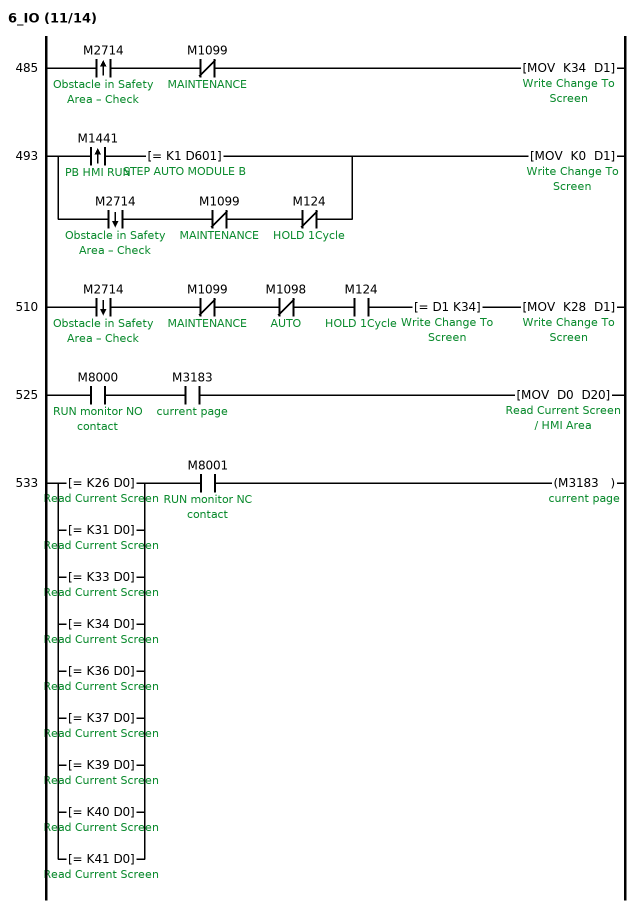
[picture p72: ladder of 6_IO, rungs at steps 485 to 533]
485   LDP     M2714  ; Obstacle in Safety Area – Check
      ANI     M1099  ; MAINTENANCE
      MOV     K34 D1  ; Write Change To Screen
493   LDP     M1441  ; PB HMI RUN
      AND=    K1 D601  ; STEP AUTO MODULE B
      LDF     M2714  ; Obstacle in Safety Area – Check
      ANI     M1099  ; MAINTENANCE
      ANI     M124  ; HOLD 1Cycle
      ORB
      MOV     K0 D1
510   LDF     M2714  ; Obstacle in Safety Area – Check
      ANI     M1099  ; MAINTENANCE
      ANI     M1098  ; AUTO
      AND     M124  ; HOLD 1Cycle
      AND=    D1 K34  ; Write Change To Screen
      MOV     K28 D1
525   LD      M8000  ; RUN monitor NO contact
      AND     M3183  ; current page
      MOV     D0 D20  ; Read Current Screen / HMI Area
533   LD=     K26 D0  ; Read Current Screen
      OR=     K31 D0  ; Read Current Screen
      OR=     K33 D0  ; Read Current Screen
      OR=     K34 D0  ; Read Current Screen
      OR=     K36 D0  ; Read Current Screen
      OR=     K37 D0  ; Read Current Screen
      OR=     K39 D0  ; Read Current Screen
      OR=     K40 D0  ; Read Current Screen
      OR=     K41 D0  ; Read Current Screen
      AND     M8001  ; RUN monitor NC contact
      OUT     M3183  ; current page
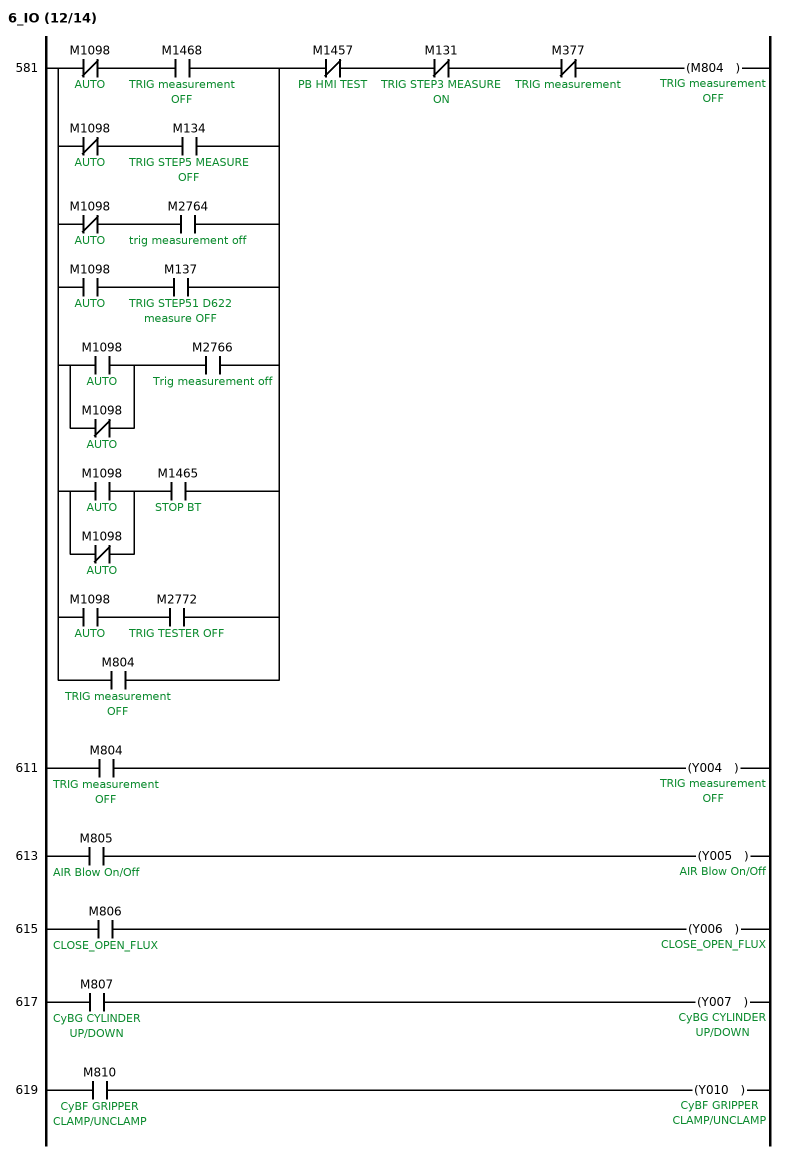
581   LDI     M1098  ; AUTO
      AND     M1468  ; TRIG measurement OFF
      LDI     M1098  ; AUTO
      AND     M134  ; TRIG STEP5 MEASURE OFF
      ORB
      LDI     M1098  ; AUTO
      AND     M2764  ; trig measurement off
      ORB
      LD      M1098  ; AUTO
      AND     M137  ; TRIG STEP51 D622 measure OFF
      ORB
      LD      M1098  ; AUTO
      ORI     M1098  ; AUTO
      AND     M2766  ; Trig measurement off
      ORB
      LD      M1098  ; AUTO
      ORI     M1098  ; AUTO
      AND     M1465  ; STOP BT
      ORB
      LD      M1098  ; AUTO
      AND     M2772  ; TRIG TESTER OFF
      ORB
      OR      M804  ; TRIG measurement OFF
      ANI     M1457  ; PB HMI TEST
      ANI     M131  ; TRIG STEP3 MEASURE ON
      ANI     M377  ; TRIG measurement
      OUT     M804  ; TRIG measurement OFF
611   LD      M804  ; TRIG measurement OFF
      OUT     Y004  ; TRIG measurement OFF
613   LD      M805  ; AIR Blow On/Off
      OUT     Y005  ; AIR Blow On/Off
615   LD      M806  ; CLOSE_OPEN_FLUX
      OUT     Y006  ; CLOSE_OPEN_FLUX
617   LD      M807  ; CyBG CYLINDER UP/DOWN
      OUT     Y007  ; CyBG CYLINDER UP/DOWN
619   LD      M810  ; CyBF GRIPPER CLAMP/UNCLAMP
      OUT     Y010  ; CyBF GRIPPER CLAMP/UNCLAMP
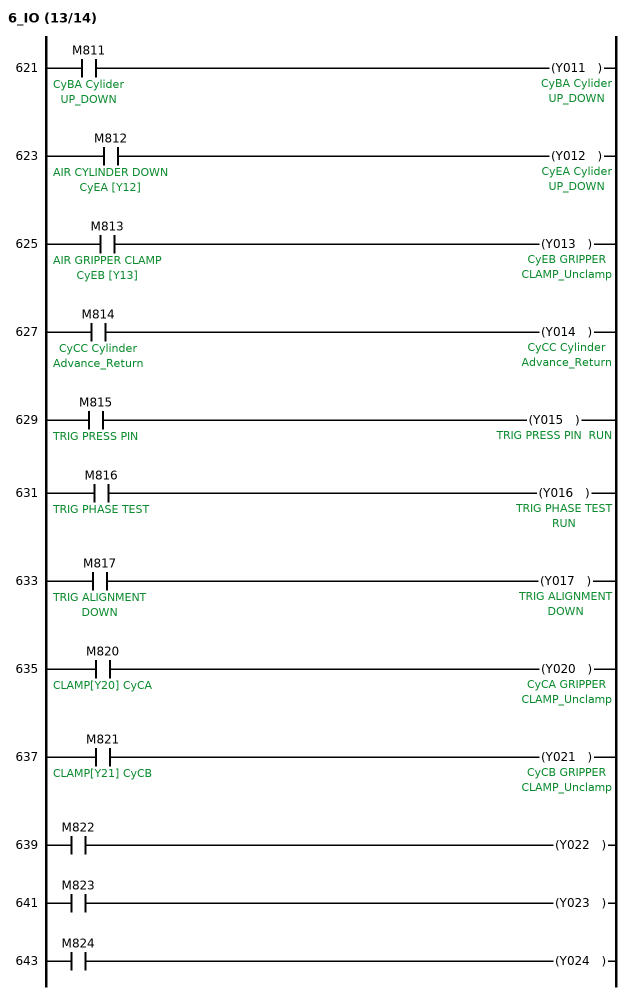
621   LD      M811  ; CyBA Cylider UP_DOWN
      OUT     Y011  ; CyBA Cylider UP_DOWN
623   LD      M812  ; AIR CYLINDER DOWN CyEA [Y12]
      OUT     Y012  ; CyEA Cylider UP_DOWN
625   LD      M813  ; AIR GRIPPER CLAMP CyEB [Y13]
      OUT     Y013  ; CyEB GRIPPER CLAMP_Unclamp
627   LD      M814  ; CyCC Cylinder Advance_Return
      OUT     Y014  ; CyCC Cylinder Advance_Return
629   LD      M815  ; TRIG PRESS PIN
      OUT     Y015  ; TRIG PRESS PIN  RUN
631   LD      M816  ; TRIG PHASE TEST
      OUT     Y016  ; TRIG PHASE TEST  RUN
633   LD      M817  ; TRIG ALIGNMENT  DOWN
      OUT     Y017  ; TRIG ALIGNMENT  DOWN
635   LD      M820  ; CLAMP[Y20] CyCA
      OUT     Y020  ; CyCA GRIPPER CLAMP_Unclamp
637   LD      M821  ; CLAMP[Y21] CyCB
      OUT     Y021  ; CyCB GRIPPER CLAMP_Unclamp
639   LD      M822
      OUT     Y022
641   LD      M823
      OUT     Y023
643   LD      M824
      OUT     Y024
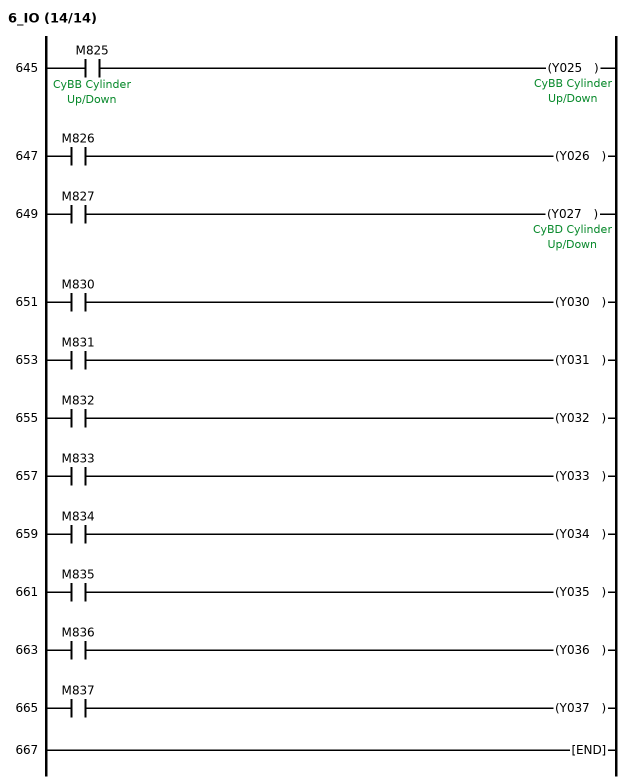
645   LD      M825  ; CyBB Cylinder Up/Down
      OUT     Y025  ; CyBB Cylinder Up/Down
647   LD      M826
      OUT     Y026
649   LD      M827
      OUT     Y027  ; CyBD Cylinder Up/Down
651   LD      M830
      OUT     Y030
653   LD      M831
      OUT     Y031
655   LD      M832
      OUT     Y032
657   LD      M833
      OUT     Y033
659   LD      M834
      OUT     Y034
661   LD      M835
      OUT     Y035
663   LD      M836
      OUT     Y036
665   LD      M837
      OUT     Y037
667   END
END_PROGRAM

PROGRAM 7_ALARM
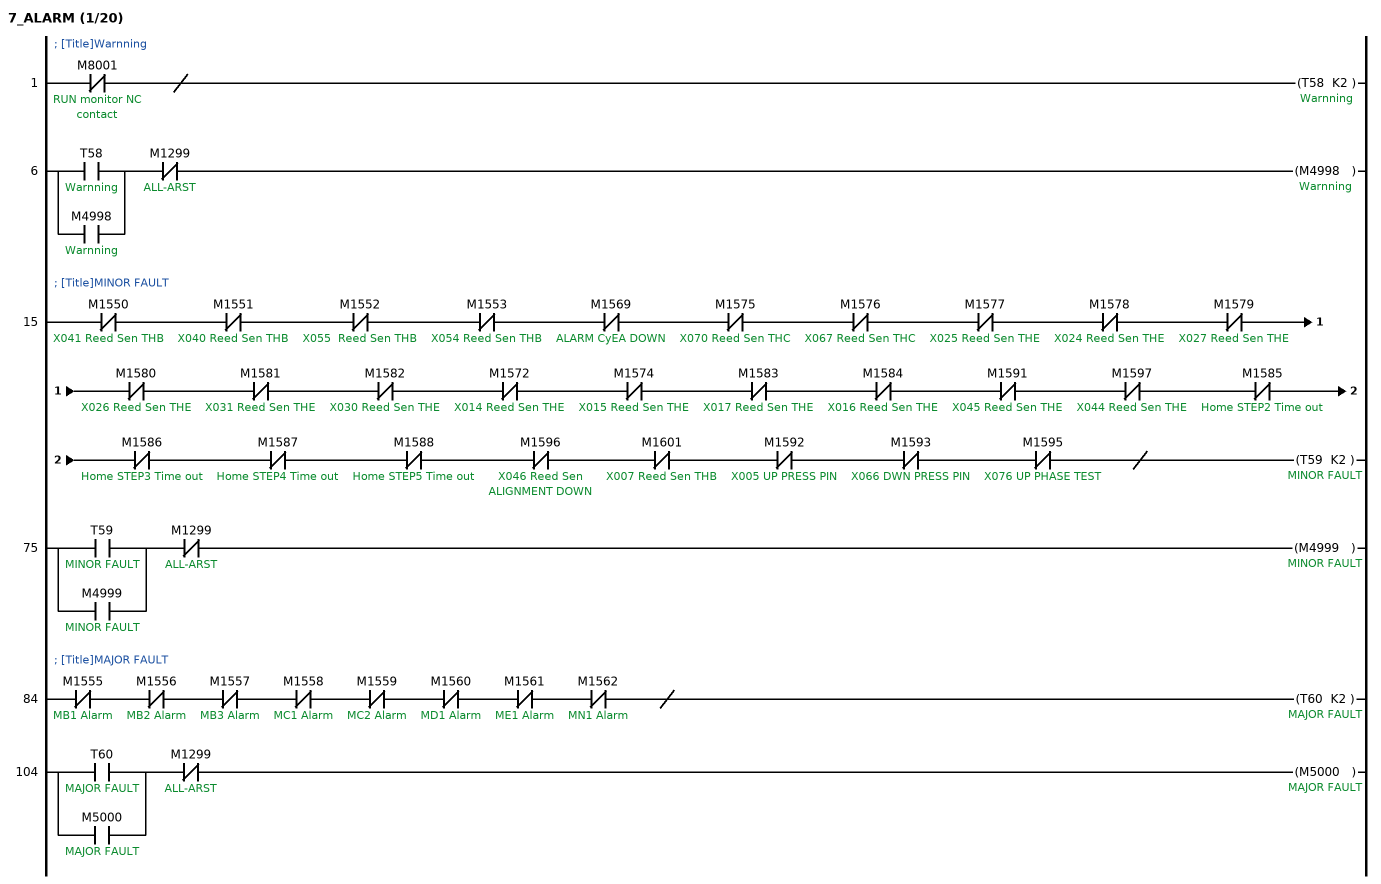
; [Title]Warnning
1     LDI     M8001  ; RUN monitor NC contact
      INV
      OUT     T58 K2  ; Warnning
6     LD      T58  ; Warnning
      OR      M4998  ; Warnning
      ANI     M1299  ; ALL-ARST
      OUT     M4998  ; Warnning
; [Title]MINOR FAULT
15    LDI     M1550  ; X041 Reed Sen THB
      ANI     M1551  ; X040 Reed Sen THB
      ANI     M1552  ; X055  Reed Sen THB
      ANI     M1553  ; X054 Reed Sen THB
      ANI     M1569  ; ALARM CyEA DOWN
      ANI     M1575  ; X070 Reed Sen THC
      ANI     M1576  ; X067 Reed Sen THC
      ANI     M1577  ; X025 Reed Sen THE
      ANI     M1578  ; X024 Reed Sen THE
      ANI     M1579  ; X027 Reed Sen THE
      ANI     M1580  ; X026 Reed Sen THE
      ANI     M1581  ; X031 Reed Sen THE
      ANI     M1582  ; X030 Reed Sen THE
      ANI     M1572  ; X014 Reed Sen THE
      ANI     M1574  ; X015 Reed Sen THE
      ANI     M1583  ; X017 Reed Sen THE
      ANI     M1584  ; X016 Reed Sen THE
      ANI     M1591  ; X045 Reed Sen THE
      ANI     M1597  ; X044 Reed Sen THE
      ANI     M1585  ; Home STEP2 Time out
      ANI     M1586  ; Home STEP3 Time out
      ANI     M1587  ; Home STEP4 Time out
      ANI     M1588  ; Home STEP5 Time out
      ANI     M1596  ; X046 Reed Sen ALIGNMENT DOWN
      ANI     M1601  ; X007 Reed Sen THB
      ANI     M1592  ; X005 UP PRESS PIN
      ANI     M1593  ; X066 DWN PRESS PIN
      ANI     M1595  ; X076 UP PHASE TEST
      INV
      OUT     T59 K2  ; MINOR FAULT
75    LD      T59  ; MINOR FAULT
      OR      M4999  ; MINOR FAULT
      ANI     M1299  ; ALL-ARST
      OUT     M4999  ; MINOR FAULT
; [Title]MAJOR FAULT
84    LDI     M1555  ; MB1 Alarm
      ANI     M1556  ; MB2 Alarm
      ANI     M1557  ; MB3 Alarm
      ANI     M1558  ; MC1 Alarm
      ANI     M1559  ; MC2 Alarm
      ANI     M1560  ; MD1 Alarm
      ANI     M1561  ; ME1 Alarm
      ANI     M1562  ; MN1 Alarm
      INV
      OUT     T60 K2  ; MAJOR FAULT
104   LD      T60  ; MAJOR FAULT
      OR      M5000  ; MAJOR FAULT
      ANI     M1299  ; ALL-ARST
      OUT     M5000  ; MAJOR FAULT
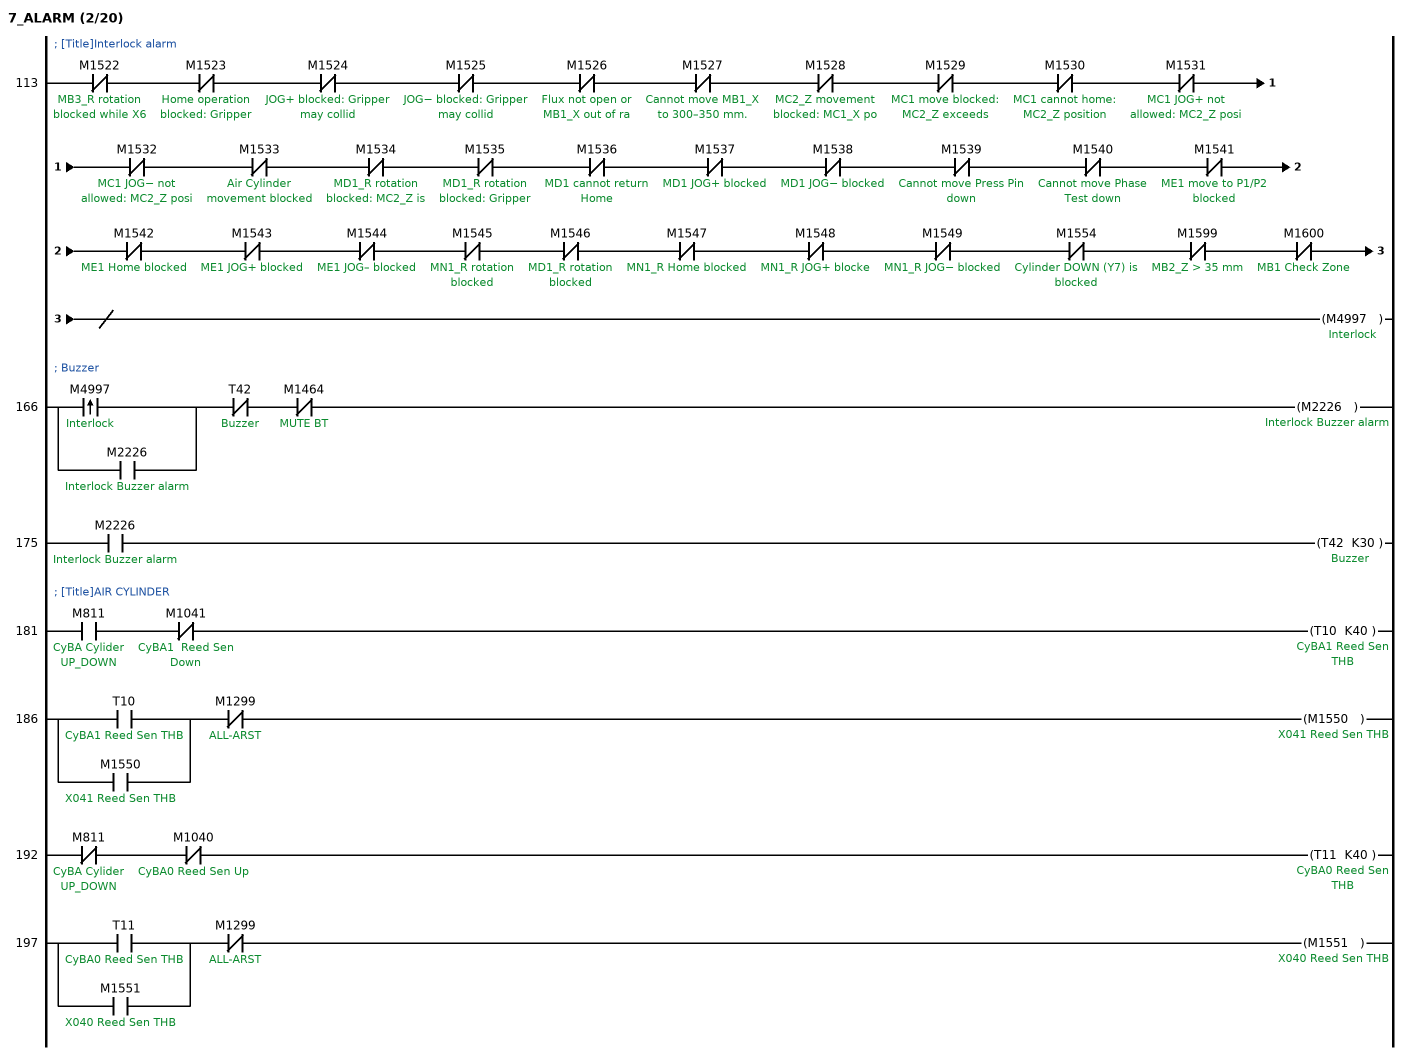
; [Title]Interlock alarm
113   LDI     M1522  ; MB3_R rotation blocked while X6
      ANI     M1523  ; Home operation blocked: Gripper
      ANI     M1524  ; JOG+ blocked: Gripper may collid
      ANI     M1525  ; JOG− blocked: Gripper may collid
      ANI     M1526  ; Flux not open or MB1_X out of ra
      ANI     M1527  ; Cannot move MB1_X to 300–350 mm.
      ANI     M1528  ; MC2_Z movement blocked: MC1_X po
      ANI     M1529  ; MC1 move blocked: MC2_Z exceeds
      ANI     M1530  ; MC1 cannot home: MC2_Z position
      ANI     M1531  ; MC1 JOG+ not allowed: MC2_Z posi
      ANI     M1532  ; MC1 JOG− not allowed: MC2_Z posi
      ANI     M1533  ; Air Cylinder movement blocked
      ANI     M1534  ; MD1_R rotation blocked: MC2_Z is
      ANI     M1535  ; MD1_R rotation blocked: Gripper
      ANI     M1536  ; MD1 cannot return Home
      ANI     M1537  ; MD1 JOG+ blocked
      ANI     M1538  ; MD1 JOG− blocked
      ANI     M1539  ; Cannot move Press Pin down
      ANI     M1540  ; Cannot move Phase Test down
      ANI     M1541  ; ME1 move to P1/P2 blocked
      ANI     M1542  ; ME1 Home blocked
      ANI     M1543  ; ME1 JOG+ blocked
      ANI     M1544  ; ME1 JOG– blocked
      ANI     M1545  ; MN1_R rotation blocked
      ANI     M1546  ; MD1_R rotation blocked
      ANI     M1547  ; MN1_R Home blocked
      ANI     M1548  ; MN1_R JOG+ blocke
      ANI     M1549  ; MN1_R JOG− blocked
      ANI     M1554  ; Cylinder DOWN (Y7) is blocked
      ANI     M1599  ; MB2_Z > 35 mm
      ANI     M1600  ; MB1 Check Zone
      INV
      OUT     M4997  ; Interlock
; Buzzer
166   LDP     M4997  ; Interlock
      OR      M2226  ; Interlock Buzzer alarm
      ANI     T42  ; Buzzer
      ANI     M1464  ; MUTE BT
      OUT     M2226  ; Interlock Buzzer alarm
175   LD      M2226  ; Interlock Buzzer alarm
      OUT     T42 K30  ; Buzzer
; [Title]AIR CYLINDER
181   LD      M811  ; CyBA Cylider UP_DOWN
      ANI     M1041  ; CyBA1  Reed Sen Down
      OUT     T10 K40  ; CyBA1 Reed Sen THB
186   LD      T10  ; CyBA1 Reed Sen THB
      OR      M1550  ; X041 Reed Sen THB
      ANI     M1299  ; ALL-ARST
      OUT     M1550  ; X041 Reed Sen THB
192   LDI     M811  ; CyBA Cylider UP_DOWN
      ANI     M1040  ; CyBA0 Reed Sen Up
      OUT     T11 K40  ; CyBA0 Reed Sen THB
197   LD      T11  ; CyBA0 Reed Sen THB
      OR      M1551  ; X040 Reed Sen THB
      ANI     M1299  ; ALL-ARST
      OUT     M1551  ; X040 Reed Sen THB
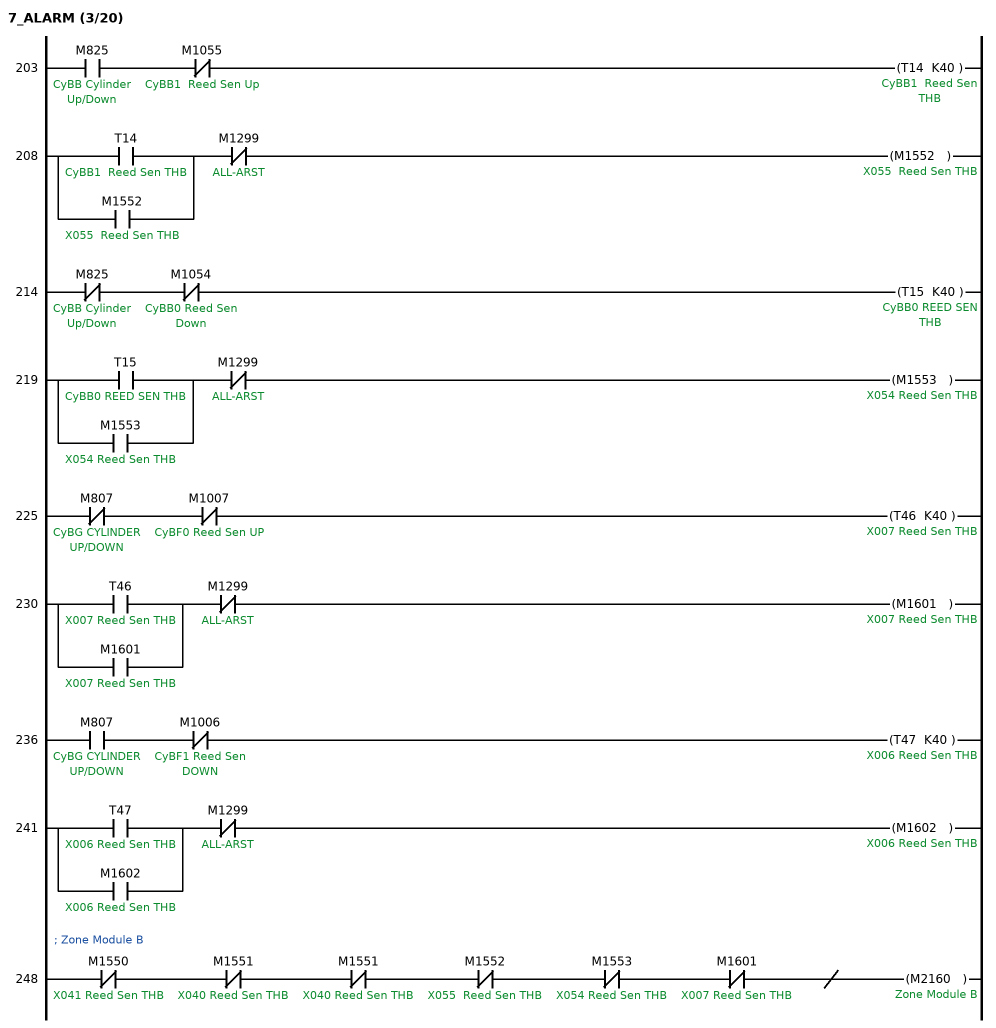
203   LD      M825  ; CyBB Cylinder Up/Down
      ANI     M1055  ; CyBB1  Reed Sen Up
      OUT     T14 K40  ; CyBB1  Reed Sen THB
208   LD      T14  ; CyBB1  Reed Sen THB
      OR      M1552  ; X055  Reed Sen THB
      ANI     M1299  ; ALL-ARST
      OUT     M1552  ; X055  Reed Sen THB
214   LDI     M825  ; CyBB Cylinder Up/Down
      ANI     M1054  ; CyBB0 Reed Sen Down
      OUT     T15 K40  ; CyBB0 REED SEN THB
219   LD      T15  ; CyBB0 REED SEN THB
      OR      M1553  ; X054 Reed Sen THB
      ANI     M1299  ; ALL-ARST
      OUT     M1553  ; X054 Reed Sen THB
225   LDI     M807  ; CyBG CYLINDER UP/DOWN
      ANI     M1007  ; CyBF0 Reed Sen UP
      OUT     T46 K40  ; X007 Reed Sen THB
230   LD      T46  ; X007 Reed Sen THB
      OR      M1601  ; X007 Reed Sen THB
      ANI     M1299  ; ALL-ARST
      OUT     M1601  ; X007 Reed Sen THB
236   LD      M807  ; CyBG CYLINDER UP/DOWN
      ANI     M1006  ; CyBF1 Reed Sen DOWN
      OUT     T47 K40  ; X006 Reed Sen THB
241   LD      T47  ; X006 Reed Sen THB
      OR      M1602  ; X006 Reed Sen THB
      ANI     M1299  ; ALL-ARST
      OUT     M1602  ; X006 Reed Sen THB
; Zone Module B
248   LDI     M1550  ; X041 Reed Sen THB
      ANI     M1551  ; X040 Reed Sen THB
      ANI     M1551  ; X040 Reed Sen THB
      ANI     M1552  ; X055  Reed Sen THB
      ANI     M1553  ; X054 Reed Sen THB
      ANI     M1601  ; X007 Reed Sen THB
      INV
      OUT     M2160  ; Zone Module B
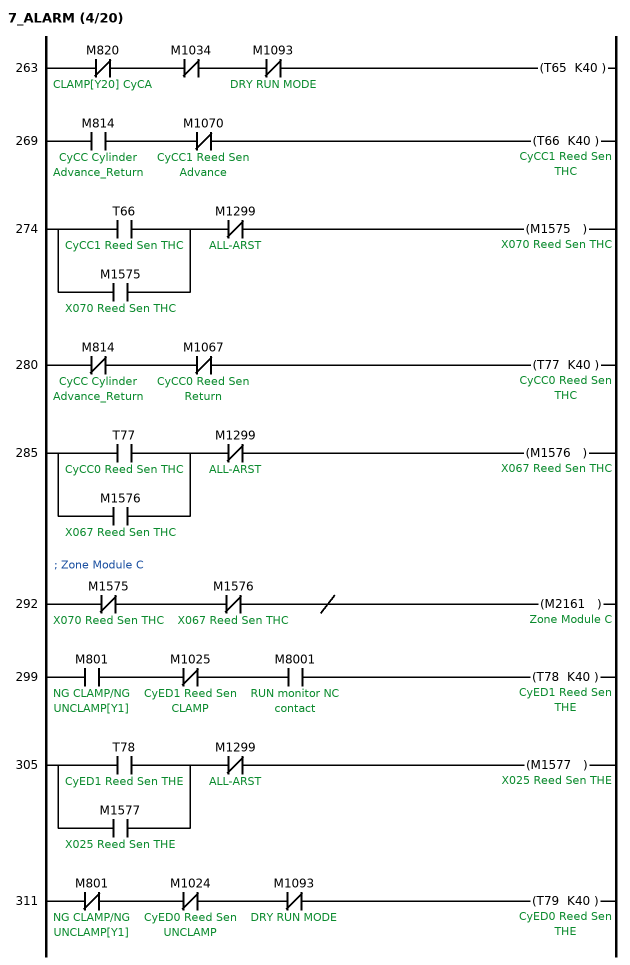
263   LDI     M820  ; CLAMP[Y20] CyCA
      ANI     M1034
      ANI     M1093  ; DRY RUN MODE
      OUT     T65 K40
269   LD      M814  ; CyCC Cylinder Advance_Return
      ANI     M1070  ; CyCC1 Reed Sen  Advance
      OUT     T66 K40  ; CyCC1 Reed Sen THC
274   LD      T66  ; CyCC1 Reed Sen THC
      OR      M1575  ; X070 Reed Sen THC
      ANI     M1299  ; ALL-ARST
      OUT     M1575  ; X070 Reed Sen THC
280   LDI     M814  ; CyCC Cylinder Advance_Return
      ANI     M1067  ; CyCC0 Reed Sen Return
      OUT     T77 K40  ; CyCC0 Reed Sen THC
285   LD      T77  ; CyCC0 Reed Sen THC
      OR      M1576  ; X067 Reed Sen THC
      ANI     M1299  ; ALL-ARST
      OUT     M1576  ; X067 Reed Sen THC
; Zone Module C
292   LDI     M1575  ; X070 Reed Sen THC
      ANI     M1576  ; X067 Reed Sen THC
      INV
      OUT     M2161  ; Zone Module C
299   LD      M801  ; NG CLAMP/NG UNCLAMP[Y1]
      ANI     M1025  ; CyED1 Reed Sen CLAMP
      AND     M8001  ; RUN monitor NC contact
      OUT     T78 K40  ; CyED1 Reed Sen THE
305   LD      T78  ; CyED1 Reed Sen THE
      OR      M1577  ; X025 Reed Sen THE
      ANI     M1299  ; ALL-ARST
      OUT     M1577  ; X025 Reed Sen THE
311   LDI     M801  ; NG CLAMP/NG UNCLAMP[Y1]
      ANI     M1024  ; CyED0 Reed Sen UNCLAMP
      ANI     M1093  ; DRY RUN MODE
      OUT     T79 K40  ; CyED0 Reed Sen THE
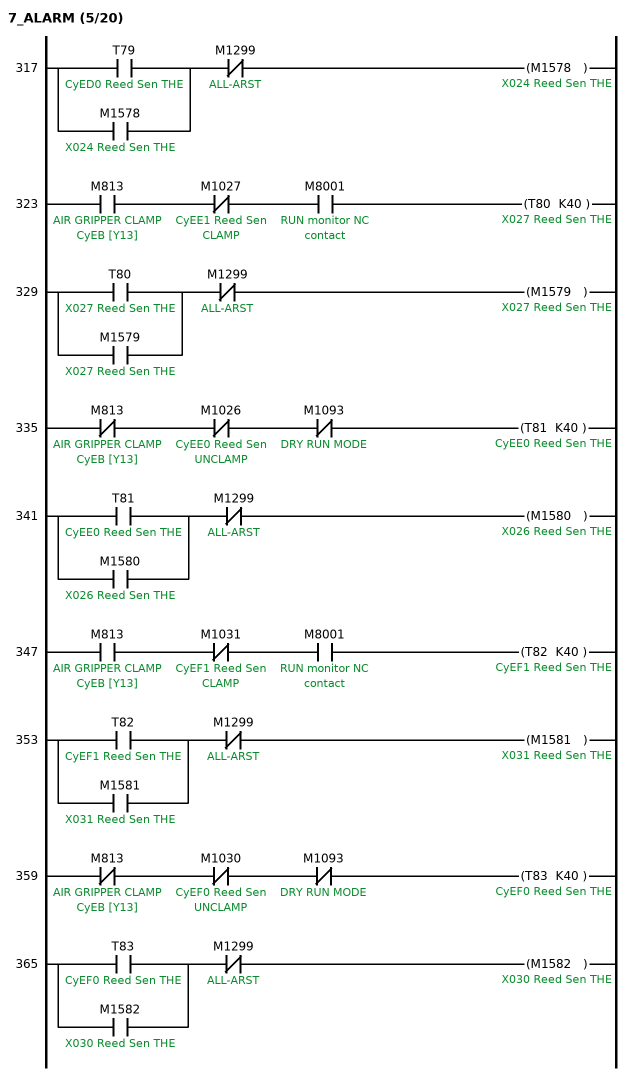
317   LD      T79  ; CyED0 Reed Sen THE
      OR      M1578  ; X024 Reed Sen THE
      ANI     M1299  ; ALL-ARST
      OUT     M1578  ; X024 Reed Sen THE
323   LD      M813  ; AIR GRIPPER CLAMP CyEB [Y13]
      ANI     M1027  ; CyEE1 Reed Sen CLAMP
      AND     M8001  ; RUN monitor NC contact
      OUT     T80 K40  ; X027 Reed Sen THE
329   LD      T80  ; X027 Reed Sen THE
      OR      M1579  ; X027 Reed Sen THE
      ANI     M1299  ; ALL-ARST
      OUT     M1579  ; X027 Reed Sen THE
335   LDI     M813  ; AIR GRIPPER CLAMP CyEB [Y13]
      ANI     M1026  ; CyEE0 Reed Sen UNCLAMP
      ANI     M1093  ; DRY RUN MODE
      OUT     T81 K40  ; CyEE0 Reed Sen THE
341   LD      T81  ; CyEE0 Reed Sen THE
      OR      M1580  ; X026 Reed Sen THE
      ANI     M1299  ; ALL-ARST
      OUT     M1580  ; X026 Reed Sen THE
347   LD      M813  ; AIR GRIPPER CLAMP CyEB [Y13]
      ANI     M1031  ; CyEF1 Reed Sen CLAMP
      AND     M8001  ; RUN monitor NC contact
      OUT     T82 K40  ; CyEF1 Reed Sen THE
353   LD      T82  ; CyEF1 Reed Sen THE
      OR      M1581  ; X031 Reed Sen THE
      ANI     M1299  ; ALL-ARST
      OUT     M1581  ; X031 Reed Sen THE
359   LDI     M813  ; AIR GRIPPER CLAMP CyEB [Y13]
      ANI     M1030  ; CyEF0 Reed Sen UNCLAMP
      ANI     M1093  ; DRY RUN MODE
      OUT     T83 K40  ; CyEF0 Reed Sen THE
365   LD      T83  ; CyEF0 Reed Sen THE
      OR      M1582  ; X030 Reed Sen THE
      ANI     M1299  ; ALL-ARST
      OUT     M1582  ; X030 Reed Sen THE
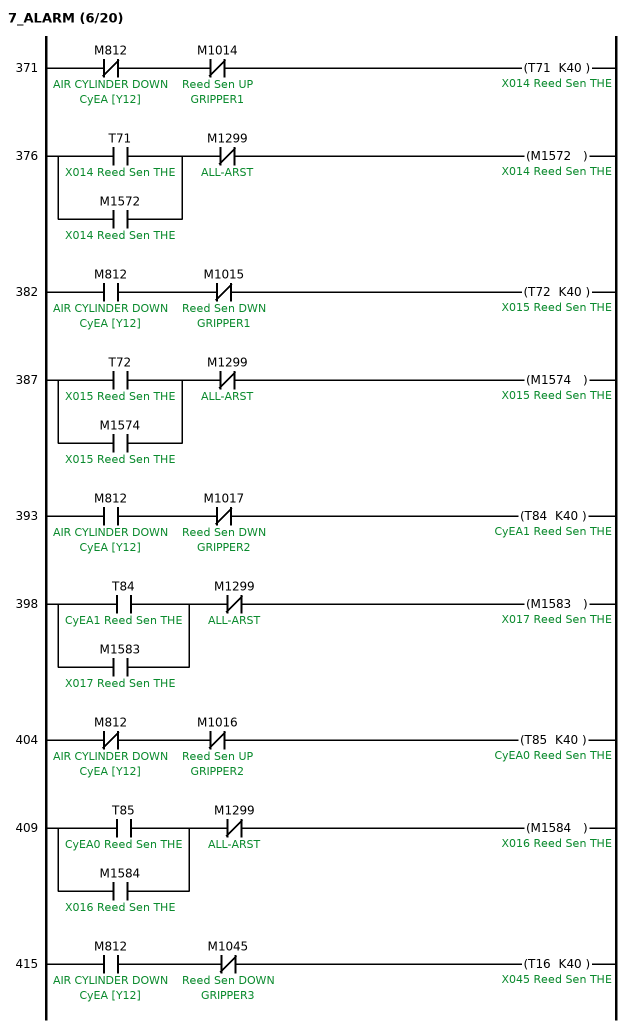
371   LDI     M812  ; AIR CYLINDER DOWN CyEA [Y12]
      ANI     M1014  ; Reed Sen UP GRIPPER1
      OUT     T71 K40  ; X014 Reed Sen THE
376   LD      T71  ; X014 Reed Sen THE
      OR      M1572  ; X014 Reed Sen THE
      ANI     M1299  ; ALL-ARST
      OUT     M1572  ; X014 Reed Sen THE
382   LD      M812  ; AIR CYLINDER DOWN CyEA [Y12]
      ANI     M1015  ; Reed Sen DWN GRIPPER1
      OUT     T72 K40  ; X015 Reed Sen THE
387   LD      T72  ; X015 Reed Sen THE
      OR      M1574  ; X015 Reed Sen THE
      ANI     M1299  ; ALL-ARST
      OUT     M1574  ; X015 Reed Sen THE
393   LD      M812  ; AIR CYLINDER DOWN CyEA [Y12]
      ANI     M1017  ; Reed Sen DWN GRIPPER2
      OUT     T84 K40  ; CyEA1 Reed Sen THE
398   LD      T84  ; CyEA1 Reed Sen THE
      OR      M1583  ; X017 Reed Sen THE
      ANI     M1299  ; ALL-ARST
      OUT     M1583  ; X017 Reed Sen THE
404   LDI     M812  ; AIR CYLINDER DOWN CyEA [Y12]
      ANI     M1016  ; Reed Sen UP GRIPPER2
      OUT     T85 K40  ; CyEA0 Reed Sen THE
409   LD      T85  ; CyEA0 Reed Sen THE
      OR      M1584  ; X016 Reed Sen THE
      ANI     M1299  ; ALL-ARST
      OUT     M1584  ; X016 Reed Sen THE
415   LD      M812  ; AIR CYLINDER DOWN CyEA [Y12]
      ANI     M1045  ; Reed Sen DOWN GRIPPER3
      OUT     T16 K40  ; X045 Reed Sen THE
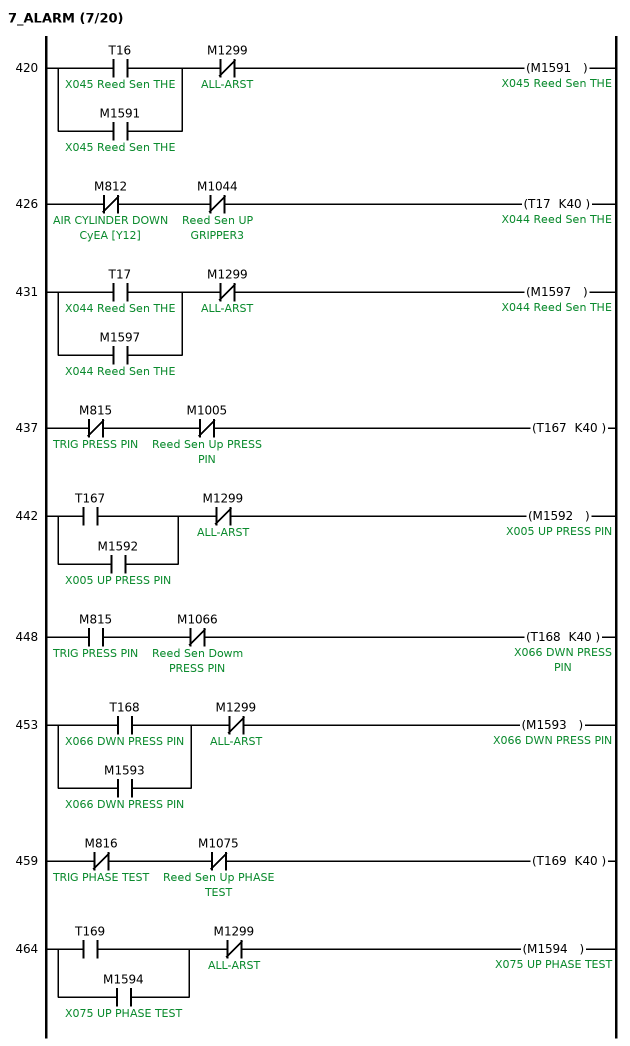
420   LD      T16  ; X045 Reed Sen THE
      OR      M1591  ; X045 Reed Sen THE
      ANI     M1299  ; ALL-ARST
      OUT     M1591  ; X045 Reed Sen THE
426   LDI     M812  ; AIR CYLINDER DOWN CyEA [Y12]
      ANI     M1044  ; Reed Sen UP GRIPPER3
      OUT     T17 K40  ; X044 Reed Sen THE
431   LD      T17  ; X044 Reed Sen THE
      OR      M1597  ; X044 Reed Sen THE
      ANI     M1299  ; ALL-ARST
      OUT     M1597  ; X044 Reed Sen THE
437   LDI     M815  ; TRIG PRESS PIN
      ANI     M1005  ; Reed Sen Up PRESS PIN
      OUT     T167 K40
442   LD      T167
      OR      M1592  ; X005 UP PRESS PIN
      ANI     M1299  ; ALL-ARST
      OUT     M1592  ; X005 UP PRESS PIN
448   LD      M815  ; TRIG PRESS PIN
      ANI     M1066  ; Reed Sen Dowm PRESS PIN
      OUT     T168 K40  ; X066 DWN PRESS PIN
453   LD      T168  ; X066 DWN PRESS PIN
      OR      M1593  ; X066 DWN PRESS PIN
      ANI     M1299  ; ALL-ARST
      OUT     M1593  ; X066 DWN PRESS PIN
459   LDI     M816  ; TRIG PHASE TEST
      ANI     M1075  ; Reed Sen Up PHASE TEST
      OUT     T169 K40
464   LD      T169
      OR      M1594  ; X075 UP PHASE TEST
      ANI     M1299  ; ALL-ARST
      OUT     M1594  ; X075 UP PHASE TEST
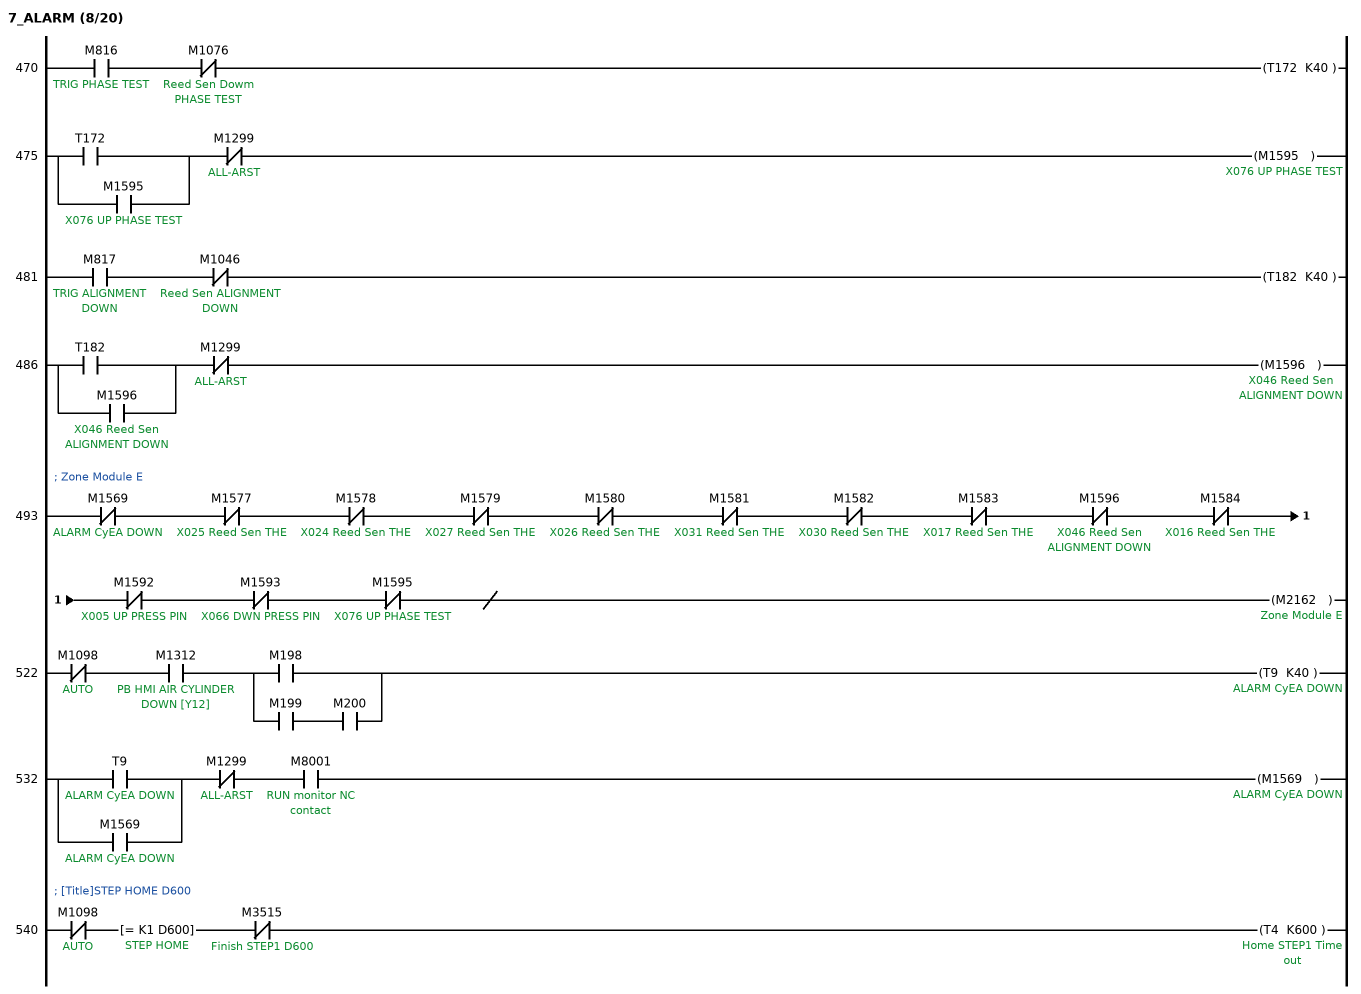
470   LD      M816  ; TRIG PHASE TEST
      ANI     M1076  ; Reed Sen Dowm PHASE TEST
      OUT     T172 K40
475   LD      T172
      OR      M1595  ; X076 UP PHASE TEST
      ANI     M1299  ; ALL-ARST
      OUT     M1595  ; X076 UP PHASE TEST
481   LD      M817  ; TRIG ALIGNMENT  DOWN
      ANI     M1046  ; Reed Sen ALIGNMENT DOWN
      OUT     T182 K40
486   LD      T182
      OR      M1596  ; X046 Reed Sen ALIGNMENT DOWN
      ANI     M1299  ; ALL-ARST
      OUT     M1596  ; X046 Reed Sen ALIGNMENT DOWN
; Zone Module E
493   LDI     M1569  ; ALARM CyEA DOWN
      ANI     M1577  ; X025 Reed Sen THE
      ANI     M1578  ; X024 Reed Sen THE
      ANI     M1579  ; X027 Reed Sen THE
      ANI     M1580  ; X026 Reed Sen THE
      ANI     M1581  ; X031 Reed Sen THE
      ANI     M1582  ; X030 Reed Sen THE
      ANI     M1583  ; X017 Reed Sen THE
      ANI     M1596  ; X046 Reed Sen ALIGNMENT DOWN
      ANI     M1584  ; X016 Reed Sen THE
      ANI     M1592  ; X005 UP PRESS PIN
      ANI     M1593  ; X066 DWN PRESS PIN
      ANI     M1595  ; X076 UP PHASE TEST
      INV
      OUT     M2162  ; Zone Module E
522   LDI     M1098  ; AUTO
      AND     M1312  ; PB HMI AIR CYLINDER DOWN [Y12]
      LD      M198
      LD      M199
      AND     M200
      ORB
      ANB
      OUT     T9 K40  ; ALARM CyEA DOWN
532   LD      T9  ; ALARM CyEA DOWN
      OR      M1569  ; ALARM CyEA DOWN
      ANI     M1299  ; ALL-ARST
      AND     M8001  ; RUN monitor NC contact
      OUT     M1569  ; ALARM CyEA DOWN
; [Title]STEP HOME D600
540   LDI     M1098  ; AUTO
      AND=    K1 D600  ; STEP HOME
      ANI     M3515  ; Finish STEP1 D600
      OUT     T4 K600  ; Home STEP1 Time out
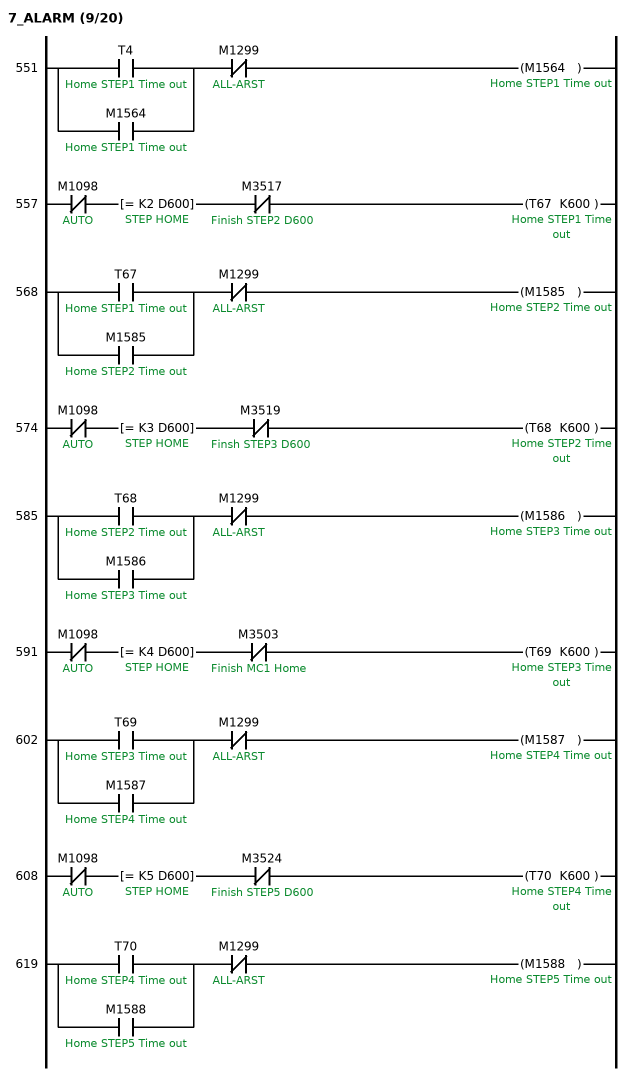
551   LD      T4  ; Home STEP1 Time out
      OR      M1564  ; Home STEP1 Time out
      ANI     M1299  ; ALL-ARST
      OUT     M1564  ; Home STEP1 Time out
557   LDI     M1098  ; AUTO
      AND=    K2 D600  ; STEP HOME
      ANI     M3517  ; Finish STEP2 D600
      OUT     T67 K600  ; Home STEP1 Time out
568   LD      T67  ; Home STEP1 Time out
      OR      M1585  ; Home STEP2 Time out
      ANI     M1299  ; ALL-ARST
      OUT     M1585  ; Home STEP2 Time out
574   LDI     M1098  ; AUTO
      AND=    K3 D600  ; STEP HOME
      ANI     M3519  ; Finsh STEP3 D600
      OUT     T68 K600  ; Home STEP2 Time out
585   LD      T68  ; Home STEP2 Time out
      OR      M1586  ; Home STEP3 Time out
      ANI     M1299  ; ALL-ARST
      OUT     M1586  ; Home STEP3 Time out
591   LDI     M1098  ; AUTO
      AND=    K4 D600  ; STEP HOME
      ANI     M3503  ; Finish MC1 Home
      OUT     T69 K600  ; Home STEP3 Time out
602   LD      T69  ; Home STEP3 Time out
      OR      M1587  ; Home STEP4 Time out
      ANI     M1299  ; ALL-ARST
      OUT     M1587  ; Home STEP4 Time out
608   LDI     M1098  ; AUTO
      AND=    K5 D600  ; STEP HOME
      ANI     M3524  ; Finish STEP5 D600
      OUT     T70 K600  ; Home STEP4 Time out
619   LD      T70  ; Home STEP4 Time out
      OR      M1588  ; Home STEP5 Time out
      ANI     M1299  ; ALL-ARST
      OUT     M1588  ; Home STEP5 Time out
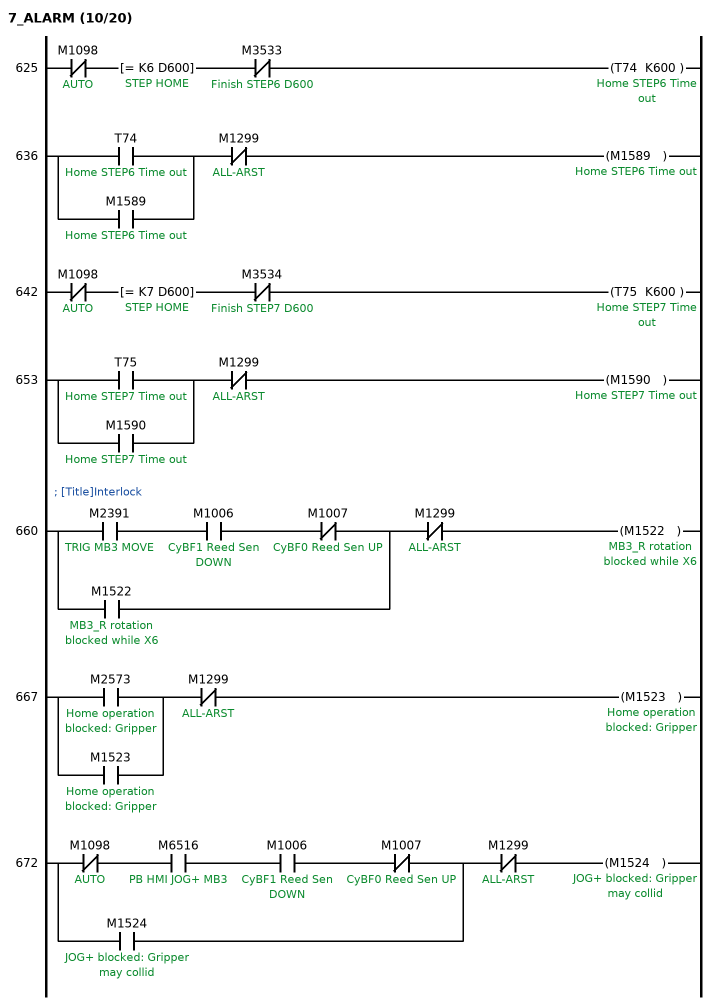
625   LDI     M1098  ; AUTO
      AND=    K6 D600  ; STEP HOME
      ANI     M3533  ; Finish STEP6 D600
      OUT     T74 K600  ; Home STEP6 Time out
636   LD      T74  ; Home STEP6 Time out
      OR      M1589  ; Home STEP6 Time out
      ANI     M1299  ; ALL-ARST
      OUT     M1589  ; Home STEP6 Time out
642   LDI     M1098  ; AUTO
      AND=    K7 D600  ; STEP HOME
      ANI     M3534  ; Finish STEP7 D600
      OUT     T75 K600  ; Home STEP7 Time out
653   LD      T75  ; Home STEP7 Time out
      OR      M1590  ; Home STEP7 Time out
      ANI     M1299  ; ALL-ARST
      OUT     M1590  ; Home STEP7 Time out
; [Title]Interlock
660   LD      M2391  ; TRIG MB3 MOVE
      AND     M1006  ; CyBF1 Reed Sen DOWN
      ANI     M1007  ; CyBF0 Reed Sen UP
      OR      M1522  ; MB3_R rotation blocked while X6
      ANI     M1299  ; ALL-ARST
      OUT     M1522  ; MB3_R rotation blocked while X6
667   LD      M2573  ; Home operation blocked: Gripper
      OR      M1523  ; Home operation blocked: Gripper
      ANI     M1299  ; ALL-ARST
      OUT     M1523  ; Home operation blocked: Gripper
672   LDI     M1098  ; AUTO
      AND     M6516  ; PB HMI JOG+ MB3
      AND     M1006  ; CyBF1 Reed Sen DOWN
      ANI     M1007  ; CyBF0 Reed Sen UP
      OR      M1524  ; JOG+ blocked: Gripper may collid
      ANI     M1299  ; ALL-ARST
      OUT     M1524  ; JOG+ blocked: Gripper may collid
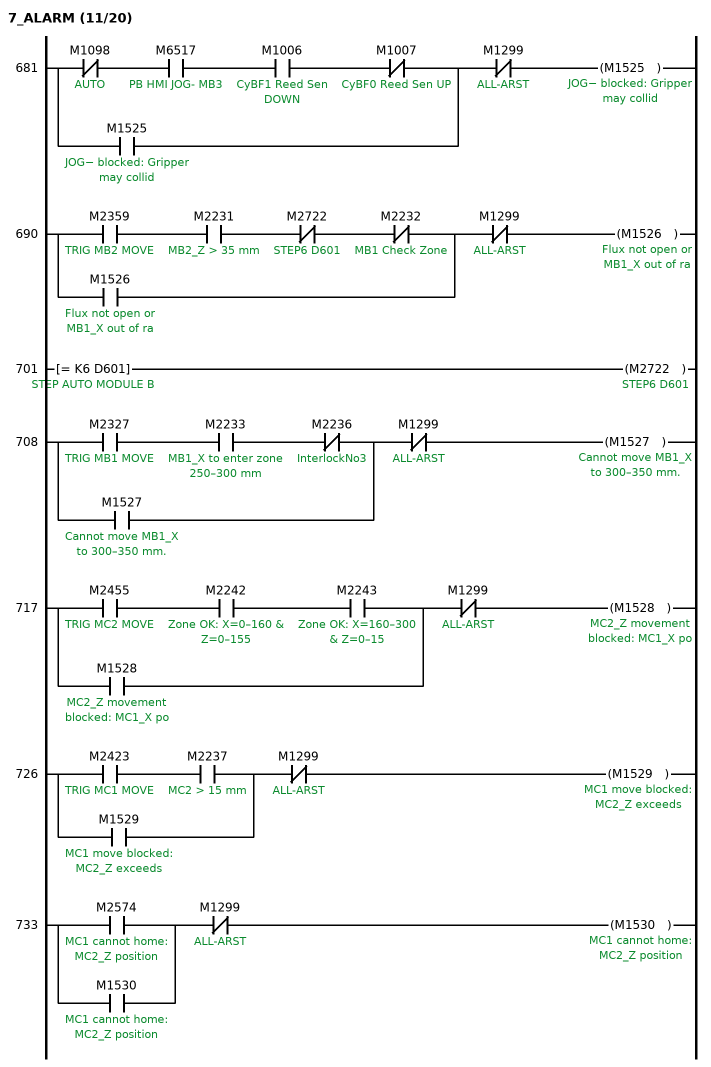
681   LDI     M1098  ; AUTO
      AND     M6517  ; PB HMI JOG- MB3
      AND     M1006  ; CyBF1 Reed Sen DOWN
      ANI     M1007  ; CyBF0 Reed Sen UP
      OR      M1525  ; JOG− blocked: Gripper may collid
      ANI     M1299  ; ALL-ARST
      OUT     M1525  ; JOG− blocked: Gripper may collid
690   LD      M2359  ; TRIG MB2 MOVE
      AND     M2231  ; MB2_Z > 35 mm
      ANI     M2722  ; STEP6 D601
      ANI     M2232  ; MB1 Check Zone
      OR      M1526  ; Flux not open or MB1_X out of ra
      ANI     M1299  ; ALL-ARST
      OUT     M1526  ; Flux not open or MB1_X out of ra
701   LD=     K6 D601  ; STEP AUTO MODULE B
      OUT     M2722  ; STEP6 D601
708   LD      M2327  ; TRIG MB1 MOVE
      AND     M2233  ; MB1_X to enter zone 250–300 mm
      ANI     M2236  ; InterlockNo3
      OR      M1527  ; Cannot move MB1_X to 300–350 mm.
      ANI     M1299  ; ALL-ARST
      OUT     M1527  ; Cannot move MB1_X to 300–350 mm.
717   LD      M2455  ; TRIG MC2 MOVE
      AND     M2242  ; Zone OK: X=0–160 & Z=0–155
      AND     M2243  ; Zone OK: X=160–300 & Z=0–15
      OR      M1528  ; MC2_Z movement blocked: MC1_X po
      ANI     M1299  ; ALL-ARST
      OUT     M1528  ; MC2_Z movement blocked: MC1_X po
726   LD      M2423  ; TRIG MC1 MOVE
      AND     M2237  ; MC2 > 15 mm
      OR      M1529  ; MC1 move blocked: MC2_Z exceeds
      ANI     M1299  ; ALL-ARST
      OUT     M1529  ; MC1 move blocked: MC2_Z exceeds
733   LD      M2574  ; MC1 cannot home: MC2_Z position
      OR      M1530  ; MC1 cannot home: MC2_Z position
      ANI     M1299  ; ALL-ARST
      OUT     M1530  ; MC1 cannot home: MC2_Z position
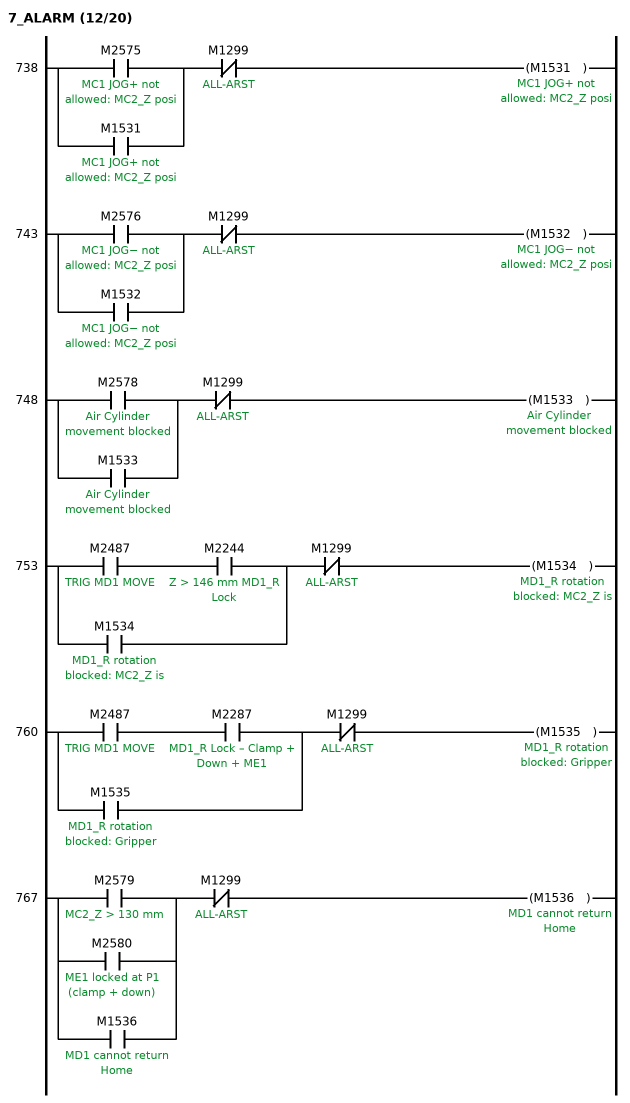
738   LD      M2575  ; MC1 JOG+ not allowed: MC2_Z posi
      OR      M1531  ; MC1 JOG+ not allowed: MC2_Z posi
      ANI     M1299  ; ALL-ARST
      OUT     M1531  ; MC1 JOG+ not allowed: MC2_Z posi
743   LD      M2576  ; MC1 JOG− not allowed: MC2_Z posi
      OR      M1532  ; MC1 JOG− not allowed: MC2_Z posi
      ANI     M1299  ; ALL-ARST
      OUT     M1532  ; MC1 JOG− not allowed: MC2_Z posi
748   LD      M2578  ; Air Cylinder movement blocked
      OR      M1533  ; Air Cylinder movement blocked
      ANI     M1299  ; ALL-ARST
      OUT     M1533  ; Air Cylinder movement blocked
753   LD      M2487  ; TRIG MD1 MOVE
      AND     M2244  ; Z > 146 mm MD1_R Lock
      OR      M1534  ; MD1_R rotation blocked: MC2_Z is
      ANI     M1299  ; ALL-ARST
      OUT     M1534  ; MD1_R rotation blocked: MC2_Z is
760   LD      M2487  ; TRIG MD1 MOVE
      AND     M2287  ; MD1_R Lock – Clamp + Down + ME1
      OR      M1535  ; MD1_R rotation blocked: Gripper
      ANI     M1299  ; ALL-ARST
      OUT     M1535  ; MD1_R rotation blocked: Gripper
767   LD      M2579  ; MC2_Z > 130 mm
      OR      M2580  ; ME1 locked at P1 (clamp + down)
      OR      M1536  ; MD1 cannot return Home
      ANI     M1299  ; ALL-ARST
      OUT     M1536  ; MD1 cannot return Home
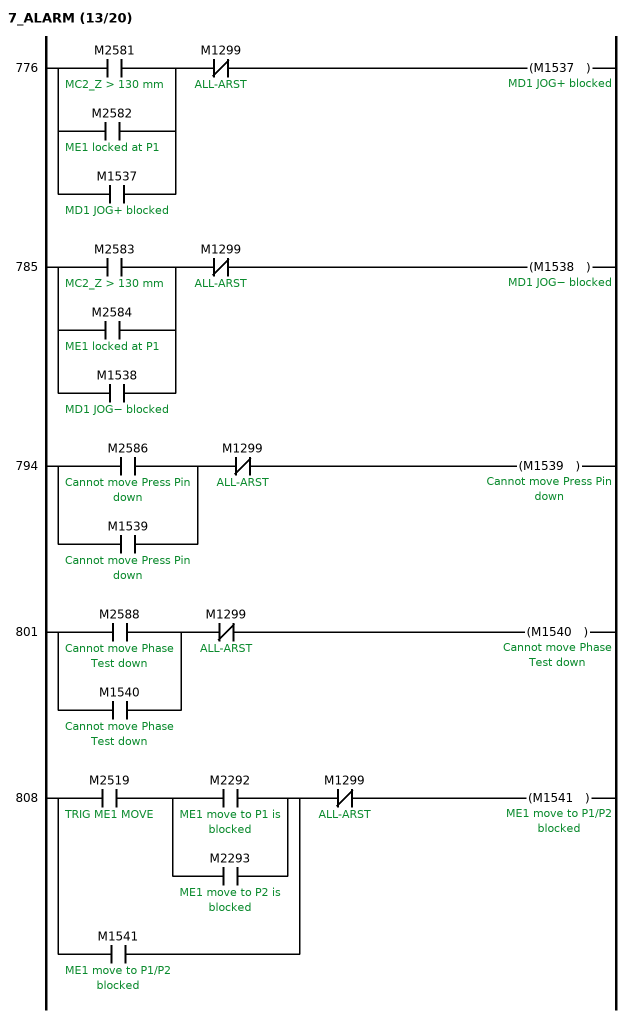
776   LD      M2581  ; MC2_Z > 130 mm
      OR      M2582  ; ME1 locked at P1
      OR      M1537  ; MD1 JOG+ blocked
      ANI     M1299  ; ALL-ARST
      OUT     M1537  ; MD1 JOG+ blocked
785   LD      M2583  ; MC2_Z > 130 mm
      OR      M2584  ; ME1 locked at P1
      OR      M1538  ; MD1 JOG− blocked
      ANI     M1299  ; ALL-ARST
      OUT     M1538  ; MD1 JOG− blocked
794   LD      M2586  ; Cannot move Press Pin down
      OR      M1539  ; Cannot move Press Pin down
      ANI     M1299  ; ALL-ARST
      OUT     M1539  ; Cannot move Press Pin down
801   LD      M2588  ; Cannot move Phase Test down
      OR      M1540  ; Cannot move Phase Test down
      ANI     M1299  ; ALL-ARST
      OUT     M1540  ; Cannot move Phase Test down
808   LD      M2519  ; TRIG ME1 MOVE
      LD      M2292  ; ME1 move to P1 is blocked
      OR      M2293  ; ME1 move to P2 is blocked
      ANB
      OR      M1541  ; ME1 move to P1/P2 blocked
      ANI     M1299  ; ALL-ARST
      OUT     M1541  ; ME1 move to P1/P2 blocked
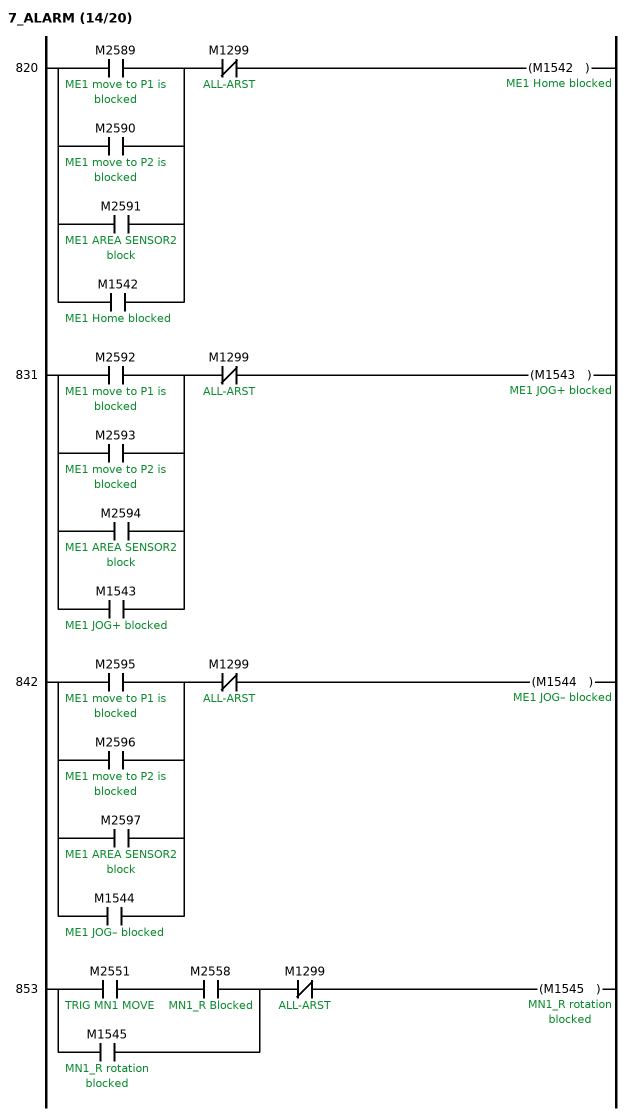
820   LD      M2589  ; ME1 move to P1 is blocked
      OR      M2590  ; ME1 move to P2 is blocked
      OR      M2591  ; ME1 AREA SENSOR2 block
      OR      M1542  ; ME1 Home blocked
      ANI     M1299  ; ALL-ARST
      OUT     M1542  ; ME1 Home blocked
831   LD      M2592  ; ME1 move to P1 is blocked
      OR      M2593  ; ME1 move to P2 is blocked
      OR      M2594  ; ME1 AREA SENSOR2 block
      OR      M1543  ; ME1 JOG+ blocked
      ANI     M1299  ; ALL-ARST
      OUT     M1543  ; ME1 JOG+ blocked
842   LD      M2595  ; ME1 move to P1 is blocked
      OR      M2596  ; ME1 move to P2 is blocked
      OR      M2597  ; ME1 AREA SENSOR2 block
      OR      M1544  ; ME1 JOG– blocked
      ANI     M1299  ; ALL-ARST
      OUT     M1544  ; ME1 JOG– blocked
853   LD      M2551  ; TRIG MN1 MOVE
      AND     M2558  ; MN1_R Blocked
      OR      M1545  ; MN1_R rotation blocked
      ANI     M1299  ; ALL-ARST
      OUT     M1545  ; MN1_R rotation blocked
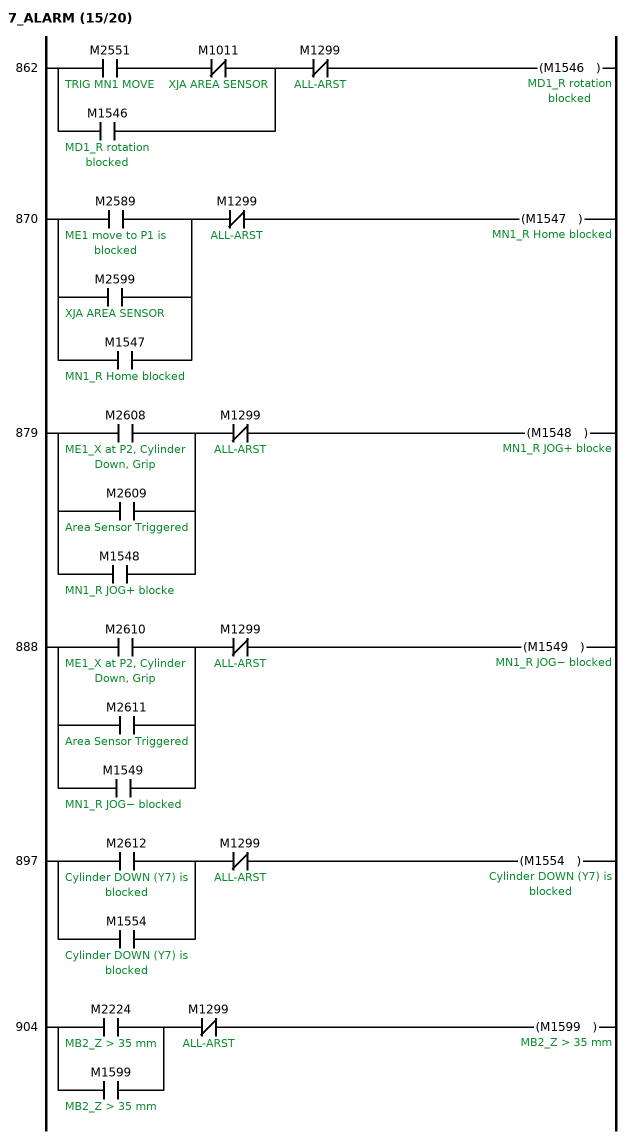
862   LD      M2551  ; TRIG MN1 MOVE
      ANI     M1011  ; XJA AREA SENSOR
      OR      M1546  ; MD1_R rotation blocked
      ANI     M1299  ; ALL-ARST
      OUT     M1546  ; MD1_R rotation blocked
870   LD      M2589  ; ME1 move to P1 is blocked
      OR      M2599  ; XJA AREA SENSOR
      OR      M1547  ; MN1_R Home blocked
      ANI     M1299  ; ALL-ARST
      OUT     M1547  ; MN1_R Home blocked
879   LD      M2608  ; ME1_X at P2, Cylinder Down, Grip
      OR      M2609  ; Area Sensor Triggered
      OR      M1548  ; MN1_R JOG+ blocke
      ANI     M1299  ; ALL-ARST
      OUT     M1548  ; MN1_R JOG+ blocke
888   LD      M2610  ; ME1_X at P2, Cylinder Down, Grip
      OR      M2611  ; Area Sensor Triggered
      OR      M1549  ; MN1_R JOG− blocked
      ANI     M1299  ; ALL-ARST
      OUT     M1549  ; MN1_R JOG− blocked
897   LD      M2612  ; Cylinder DOWN (Y7) is blocked
      OR      M1554  ; Cylinder DOWN (Y7) is blocked
      ANI     M1299  ; ALL-ARST
      OUT     M1554  ; Cylinder DOWN (Y7) is blocked
904   LD      M2224  ; MB2_Z > 35 mm
      OR      M1599  ; MB2_Z > 35 mm
      ANI     M1299  ; ALL-ARST
      OUT     M1599  ; MB2_Z > 35 mm
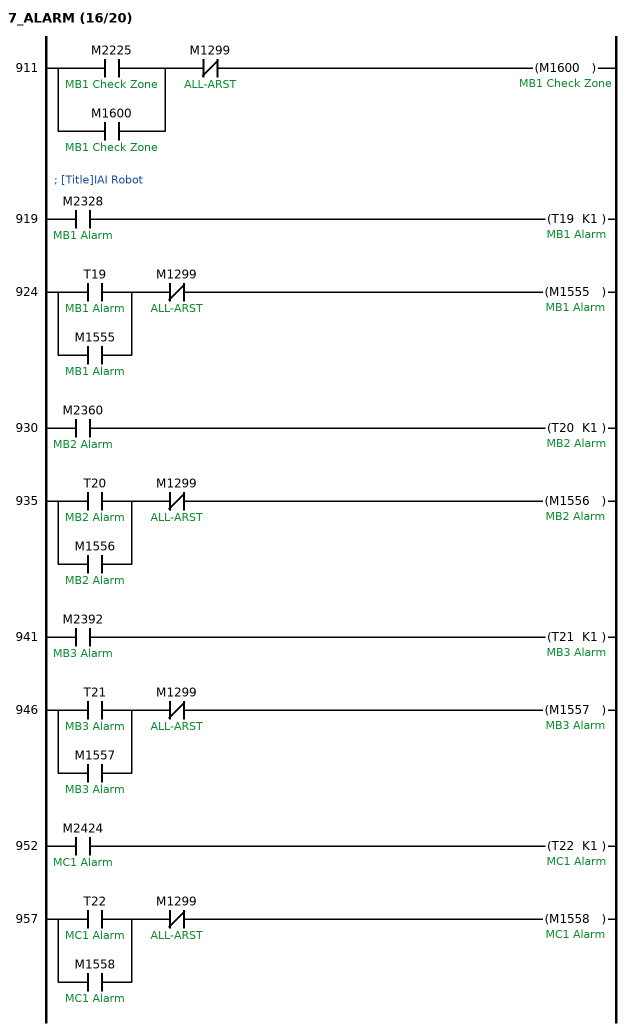
911   LD      M2225  ; MB1 Check Zone
      OR      M1600  ; MB1 Check Zone
      ANI     M1299  ; ALL-ARST
      OUT     M1600  ; MB1 Check Zone
; [Title]IAI Robot
919   LD      M2328  ; MB1 Alarm
      OUT     T19 K1  ; MB1 Alarm
924   LD      T19  ; MB1 Alarm
      OR      M1555  ; MB1 Alarm
      ANI     M1299  ; ALL-ARST
      OUT     M1555  ; MB1 Alarm
930   LD      M2360  ; MB2 Alarm
      OUT     T20 K1  ; MB2 Alarm
935   LD      T20  ; MB2 Alarm
      OR      M1556  ; MB2 Alarm
      ANI     M1299  ; ALL-ARST
      OUT     M1556  ; MB2 Alarm
941   LD      M2392  ; MB3 Alarm
      OUT     T21 K1  ; MB3 Alarm
946   LD      T21  ; MB3 Alarm
      OR      M1557  ; MB3 Alarm
      ANI     M1299  ; ALL-ARST
      OUT     M1557  ; MB3 Alarm
952   LD      M2424  ; MC1 Alarm
      OUT     T22 K1  ; MC1 Alarm
957   LD      T22  ; MC1 Alarm
      OR      M1558  ; MC1 Alarm
      ANI     M1299  ; ALL-ARST
      OUT     M1558  ; MC1 Alarm
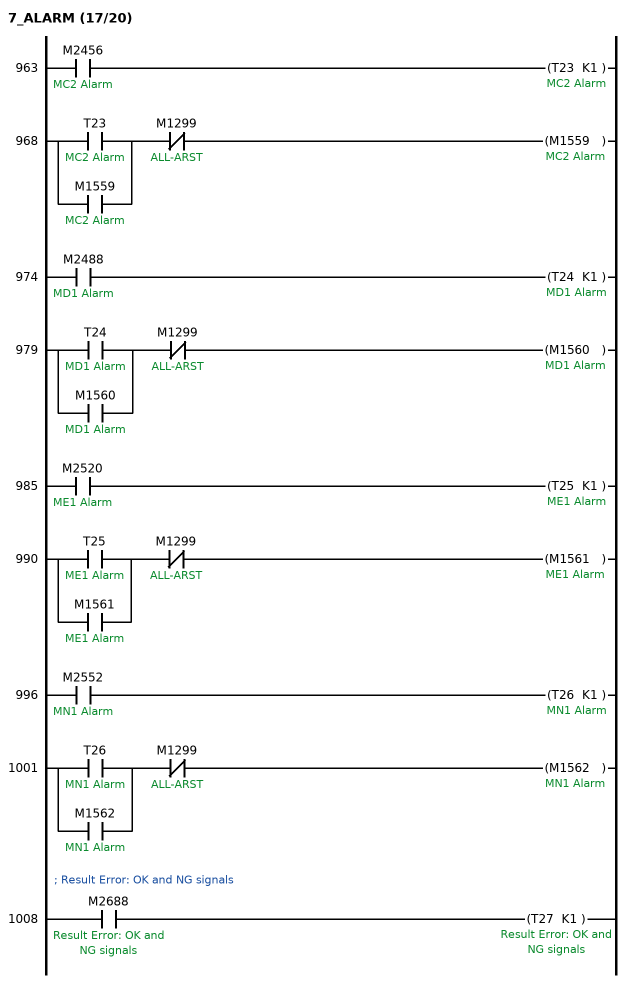
963   LD      M2456  ; MC2 Alarm
      OUT     T23 K1  ; MC2 Alarm
968   LD      T23  ; MC2 Alarm
      OR      M1559  ; MC2 Alarm
      ANI     M1299  ; ALL-ARST
      OUT     M1559  ; MC2 Alarm
974   LD      M2488  ; MD1 Alarm
      OUT     T24 K1  ; MD1 Alarm
979   LD      T24  ; MD1 Alarm
      OR      M1560  ; MD1 Alarm
      ANI     M1299  ; ALL-ARST
      OUT     M1560  ; MD1 Alarm
985   LD      M2520  ; ME1 Alarm
      OUT     T25 K1  ; ME1 Alarm
990   LD      T25  ; ME1 Alarm
      OR      M1561  ; ME1 Alarm
      ANI     M1299  ; ALL-ARST
      OUT     M1561  ; ME1 Alarm
996   LD      M2552  ; MN1 Alarm
      OUT     T26 K1  ; MN1 Alarm
1001  LD      T26  ; MN1 Alarm
      OR      M1562  ; MN1 Alarm
      ANI     M1299  ; ALL-ARST
      OUT     M1562  ; MN1 Alarm
; Result Error: OK and NG signals
1008  LD      M2688  ; Result Error: OK and NG signals
      OUT     T27 K1  ; Result Error: OK and NG signals
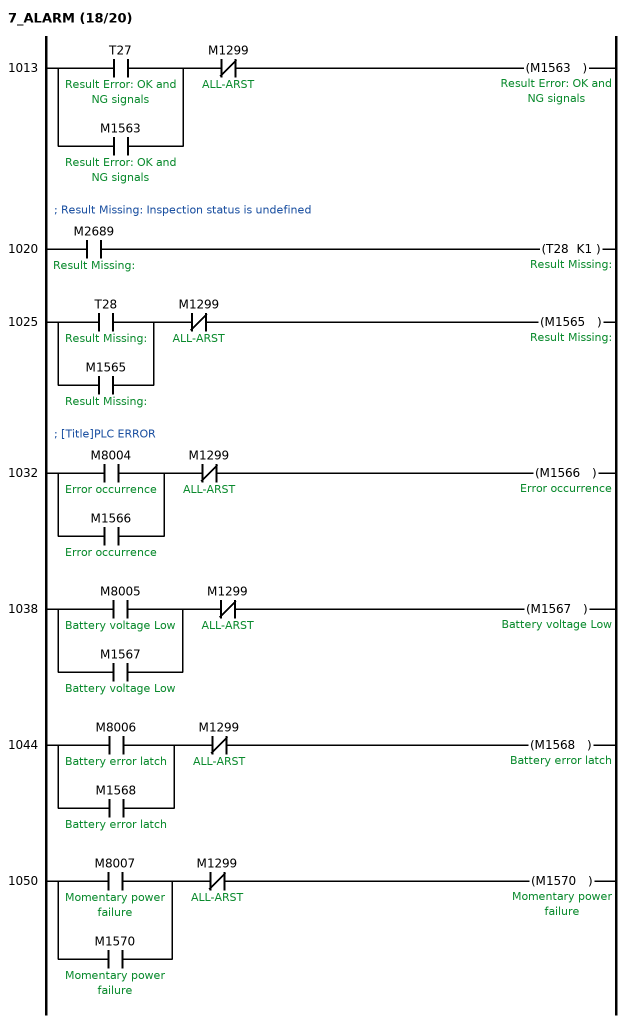
1013  LD      T27  ; Result Error: OK and NG signals
      OR      M1563  ; Result Error: OK and NG signals
      ANI     M1299  ; ALL-ARST
      OUT     M1563  ; Result Error: OK and NG signals
; Result Missing: Inspection status is undefined
1020  LD      M2689  ; Result Missing:
      OUT     T28 K1  ; Result Missing:
1025  LD      T28  ; Result Missing:
      OR      M1565  ; Result Missing:
      ANI     M1299  ; ALL-ARST
      OUT     M1565  ; Result Missing:
; [Title]PLC ERROR
1032  LD      M8004  ; Error occurrence
      OR      M1566  ; Error occurrence
      ANI     M1299  ; ALL-ARST
      OUT     M1566  ; Error occurrence
1038  LD      M8005  ; Battery voltage Low
      OR      M1567  ; Battery voltage Low
      ANI     M1299  ; ALL-ARST
      OUT     M1567  ; Battery voltage Low
1044  LD      M8006  ; Battery error latch
      OR      M1568  ; Battery error latch
      ANI     M1299  ; ALL-ARST
      OUT     M1568  ; Battery error latch
1050  LD      M8007  ; Momentary power failure
      OR      M1570  ; Momentary power failure
      ANI     M1299  ; ALL-ARST
      OUT     M1570  ; Momentary power failure
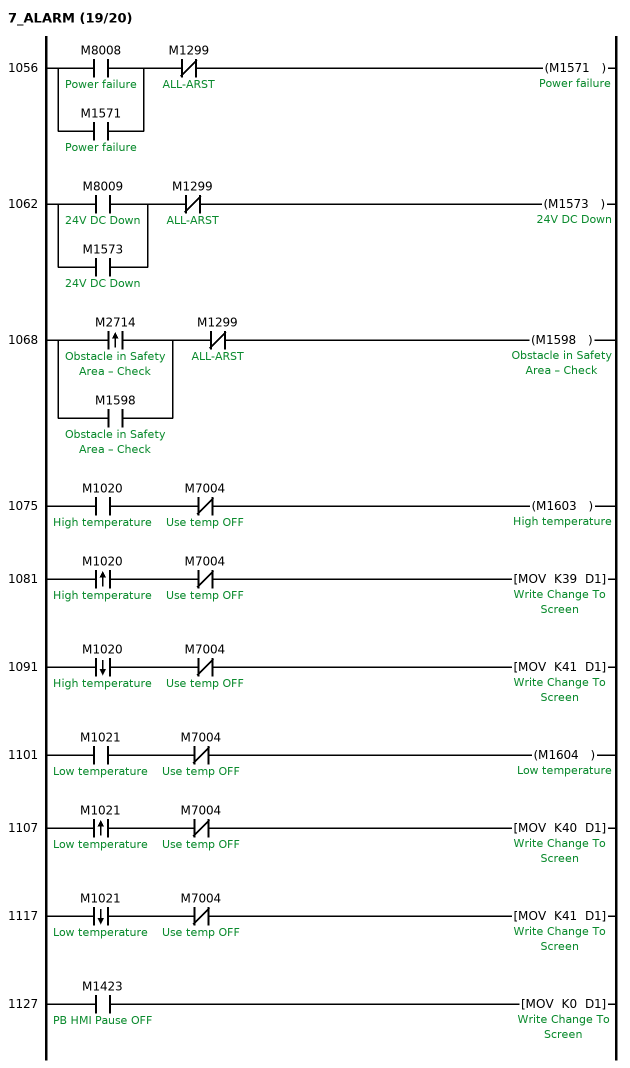
1056  LD      M8008  ; Power failure
      OR      M1571  ; Power failure
      ANI     M1299  ; ALL-ARST
      OUT     M1571  ; Power failure
1062  LD      M8009  ; 24V DC Down
      OR      M1573  ; 24V DC Down
      ANI     M1299  ; ALL-ARST
      OUT     M1573  ; 24V DC Down
1068  LDP     M2714  ; Obstacle in Safety Area – Check
      OR      M1598  ; Obstacle in Safety Area – Check
      ANI     M1299  ; ALL-ARST
      OUT     M1598  ; Obstacle in Safety Area – Check
1075  LD      M1020  ; High temperature
      ANI     M7004  ; Use temp OFF
      OUT     M1603  ; High temperature
1081  LDP     M1020  ; High temperature
      ANI     M7004  ; Use temp OFF
      MOV     K39 D1  ; Write Change To Screen
1091  LDF     M1020  ; High temperature
      ANI     M7004  ; Use temp OFF
      MOV     K41 D1
1101  LD      M1021  ; Low temperature
      ANI     M7004  ; Use temp OFF
      OUT     M1604  ; Low temperature
1107  LDP     M1021  ; Low temperature
      ANI     M7004  ; Use temp OFF
      MOV     K40 D1
1117  LDF     M1021  ; Low temperature
      ANI     M7004  ; Use temp OFF
      MOV     K41 D1
1127  LD      M1423  ; PB HMI Pause OFF
      MOV     K0 D1
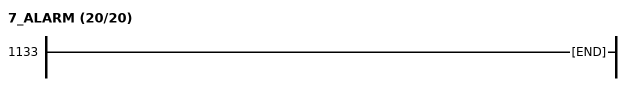
1133  END
END_PROGRAM

PROGRAM 8_ACY
